# EPICS substitutions: elioApp/Db/EL9505.substitutions
file EL9505.template { pattern
{ CHAN	, DESC		}
{ 1	, "Power OK"	}
{ 2	, "Overload"	}
}
